TYPE ST_OverCurrProtection_HWI :
STRUCT
  bEnabled  : BOOL;
  bError    : BOOL;
END_STRUCT
END_TYPE

(* stored: Version 1.1.0.1, ProductVersion 3.1.4024.12
   DUT ST_OverCurrProtection_HWI: Id {60880d17-89f5-4bbe-8cae-3ace9170e4a6} *)
